(* CODESYS project CANEcho.project

Project tree, tasks and I/O mapping:
  Device : CODESYS Control Win V3, 3S - Smart Software Solutions GmbH, order no. 305021, version 3.5.9.0
    application Application
      libraries: Standard, * (System); CANbus, 3.5.7.0 (3S - Smart Software Solutions GmbH); Common Behaviour Model Library, 0.35.9.0 (3S - Smart Software Solutions GmbH); Time and Date, 3.5.7.0 (3S - Smart Software Solutions GmbH)
      task MainTask (cyclic, interval t#20ms, priority 1) calls PLC_PRG
      program PLC_PRG [ST]
      visualisation Visualization
  text list GlobalTextList
  function block CANEcho [ST]: CyclicAction, CleanupAction, StartAction, ResetAction
*)

// Device/Application/PLC_PRG
PROGRAM PLC_PRG
VAR
	aEchoTest : ARRAY[0..ciEchoInstances-1] OF CANEcho;
	axResetBusAlarm : ARRAY[0..ciEchoInstances-1] OF BOOL;
	i : INT;
	xInit : BOOL;
END_VAR
VAR CONSTANT
	ciEchoInstances : INT := 2;
END_VAR

IF NOT xInit THEN
	FOR i := 0 TO ciEchoInstances - 1 DO
		aEchoTest[i].usiNetID := TO_USINT(i);
	END_FOR
	
	xInit := TRUE;
END_IF

FOR i := 0 TO ciEchoInstances - 1 DO
	aEchoTest[i](xResetBusAlarm := axResetBusAlarm[i]);
END_FOR

END_PROGRAM

// CANEcho
FUNCTION_BLOCK CANEcho EXTENDS CBML.LConC
VAR_INPUT
	usiNetID : USINT;
	wBaudrate : WORD := 1000;
	xSupport29bit : BOOL := TRUE;
	ctTxMessages : CAA.COUNT := 100;
	xMessageDurationTest : BOOL := TRUE;
	dwMessageDurationCOBID : DWORD := 16#701;
END_VAR
VAR_IN_OUT
	xResetBusAlarm : BOOL;
END_VAR
VAR_OUTPUT
	diagInfo : CL2.DIAGNOSIS_INFO;
	udiMessageDurationMinTimeSpan : UDINT := 16#FFFFFFFF;
	udiMessageDurationCurTimeSpan : UDINT;
	udiMessageDurationMaxTimeSpan : UDINT;
END_VAR
VAR
	hDriver : CAA.HANDLE := CAA.gc_hINVALID;
	hReceiver : CAA.HANDLE := CAA.gc_hINVALID;
	eError : CL2.ERROR;
	hRxMsg : CAA.HANDLE := CAA.gc_hINVALID;
	pRxData : POINTER TO CL2I.DATA;
	hTxMsg : CAA.HANDLE := CAA.gc_hINVALID;
	pTxData : POINTER TO CL2I.DATA;
	ctMsgLeft : CAA.COUNT;
	diMsgRecv: DINT;
	i : INT;
	
	cobId : CL2I.COBID;
	usiLen : USINT;
	x29Bit : BOOL;
	xRTR : BOOL;
	xTxFrame : BOOL;
	tkStart : CAA.TICK;
	xLastMessageDurationTest : BOOL;
	
	//Test Mode
	xEchoMessages : BOOL := TRUE;
END_VAR

SUPER^();

METHOD CyclicAction
VAR_INPUT
	itfTimingController	: CBML.ITimingController;
END_VAR
VAR_OUTPUT
	xComplete	: BOOL;
	iErrorID	: INT;
END_VAR
CL2.GetDiagnosis(hDriver, ADR(diagInfo));

{warning disable C0371}
IF xResetBusAlarm THEN
	CL2.ResetBusAlarm(hDriver);
	xResetBusAlarm := FALSE;
END_IF
{warning restore C0371}

IF (xLastMessageDurationTest <> xMessageDurationTest) THEN
	//Reset Heartbeat Test
	tkStart := 0;
	udiMessageDurationMinTimeSpan := 16#FFFFFFFF;
	udiMessageDurationCurTimeSpan := 0;
	udiMessageDurationMaxTimeSpan := 0;
END_IF

xLastMessageDurationTest := xMessageDurationTest;

REPEAT
	hRxMsg := CL2.Read(hReceiverId:=hReceiver, pctMsgLeft:=ADR(ctMsgLeft), peError:=ADR(eError));
	IF hRxMsg <> CAA.gc_hINVALID THEN
		x29Bit := CL2.Is29BitIdMessage(hMessage := hRxMsg, peError := CAA.gc_pNULL);
		xTxFrame := CL2.IsTransmitMessage(hMessage := hRxMsg, peError := CAA.gc_pNULL);
		xRTR := CL2.IsRTRMessage(hMessage := hRxMsg, peError := CAA.gc_pNULL);
		cobId := CL2.GetMessageId(hMessage := hRxMsg, peError:= CAA.gc_pNULL);
		usiLen := CL2.GetMessageLength(hMessage := hRxMsg, peError := CAA.gc_pNULL);
		pRxData := CL2.GetMessageDataPointer(hMessage := hRxMsg, peError := ADR(eError));
		diMsgRecv := diMsgRecv + 1;
		IF xEchoMessages THEN
			IF pRxData <> CAA.gc_pNULL THEN
				//echo message
				hTxMsg := CL2.CreateMessage(
						hDriver:= hDriver, 
						cobID := cobId+1, 
						usiLength := usiLen, 
						xRTR := xRTR, 
						x29BitID := x29Bit, 
						peError := ADR(eError)
				);
					
				IF hTxMsg <> CAA.gc_hINVALID THEN
					pTxData := CL2.GetMessageDataPointer(hMessage := hTxMsg, peError := ADR(eError));
					IF pTxData <> CAA.gc_pNULL AND usiLen <> 0 THEN
						FOR i := 0 TO usiLen - 1 DO
							pTxData^[i] := pRxData^[i];
						END_FOR
					END_IF
					eError := CL2.Write(hDriver:= hDriver, hMessage := hTxMsg, usiPriority := 1, xEnableSyncWindow := FALSE);
					IF eError <> CL2.ERROR.NO_ERROR THEN
						CL2.FreeMessage(hMessage := hTxMsg);
					END_IF
	
					hTxMsg := CAA.gc_hINVALID;
					pTxData := CAA.gc_pNULL;
				END_IF
			END_IF
		END_IF
		
		IF xMessageDurationTest THEN
			IF (cobId = dwMessageDurationCOBID) THEN
				IF (tkStart <> 0) THEN
					udiMessageDurationCurTimeSpan := TICKU.GetElapsedTimeInUSec(tkStart);
					IF (udiMessageDurationCurTimeSpan > udiMessageDurationMaxTimeSpan) THEN
						udiMessageDurationMaxTimeSpan := udiMessageDurationCurTimeSpan;
					ELSIF udiMessageDurationCurTimeSpan < udiMessageDurationMinTimeSpan THEN
						udiMessageDurationMinTimeSpan := udiMessageDurationCurTimeSpan;
					END_IF
				END_IF
				tkStart := TICKS.GetTick(TRUE);
			END_IF
		END_IF
		
		CL2.FreeMessage(hMessage := hRxMsg);
		hRxMsg := CAA.gc_hINVALID;
		pRxData := CAA.gc_pNULL;
	END_IF
UNTIL ctMsgLeft = 0 
END_REPEAT

CL2.GetDiagnosis(hDriver, ADR(diagInfo));
END_METHOD

METHOD CleanupAction
VAR_INPUT
	xAbortProposed	: BOOL;
	iErrorIDProposed	: INT;
END_VAR
VAR_OUTPUT
	xComplete	: BOOL;
	xAbort	: BOOL;
	iErrorID	: INT;
END_VAR
CL2.DeleteReceiver(hReceiverId := hReceiver);
hReceiver := CAA.gc_hINVALID;

CL2.DriverClose(hDriver := hDriver);
hDriver := CAA.gc_hINVALID;

xAbort := xAbortProposed;
iErrorID := iErrorIDProposed;

xComplete := TRUE;
END_METHOD

METHOD StartAction
VAR_OUTPUT
	xComplete	: BOOL;
	iErrorID	: INT;
END_VAR
hDriver:= CL2.DriverOpenH(
	usiNetId :=usiNetID, 
	uiBaudrate := wBaudrate, 
	xSupport29Bits := xSupport29bit, 
	ctMessages := ctTxMessages, 
	peError := ADR(eError)
);

IF hDriver <> CAA.gc_hINVALID THEN
	hReceiver := CL2.CreateMaskReceiver(
		hDriver:= hDriver, 
		cobIdValue := 0, 
		cobIdMask := 0, 
		xRTRValue := 0, 
		xRTRMask := 0, 
		x29BitIdValue := FALSE, 
		x29BitIdMask := NOT xSupport29bit, 
		xTransmitValue := FALSE, 
		xTransmitMask := TRUE, 
		xAlwaysNewest := FALSE, 
		eEvent := CB.EVENT.NO_EVENT, 
		xEnableSyncWindow := FALSE, 
		peError := ADR(eError)
	);
END_IF

IF hDriver = CAA.gc_hINVALID THEN
	iErrorID := 1;
ELSE
	xComplete := TRUE;
END_IF
END_METHOD

METHOD ResetAction
VAR_OUTPUT
	xComplete	: BOOL;
END_VAR
udiMessageDurationMinTimeSpan := 16#FFFFFFFF;
udiMessageDurationCurTimeSpan := 0;
udiMessageDurationMaxTimeSpan := 0;
xLastMessageDurationTest := FALSE;
xComplete := TRUE;
END_METHOD

END_FUNCTION_BLOCK

// Device/Application/Visualization
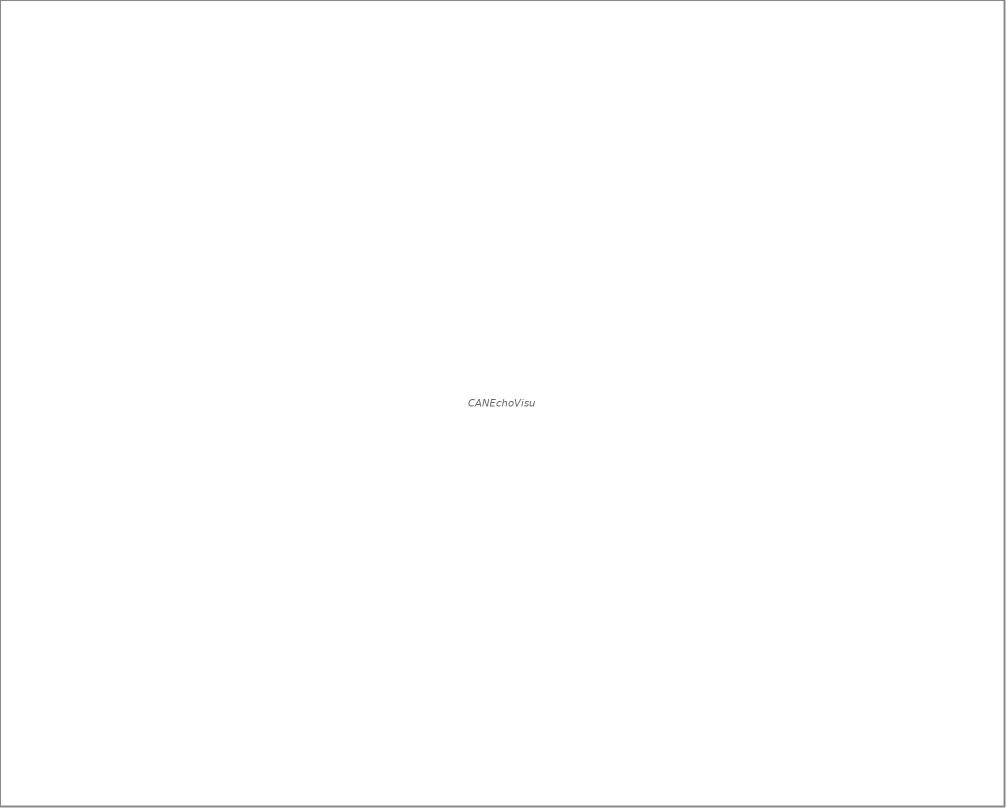
VISUALIZATION Visualization  // 1006x808
    TabControl (0,0 1004x806)
        shows CANEchoVisu(echoFB := PLC_PRG.aEchoTest[0])
        shows CANEchoVisu(echoFB := PLC_PRG.aEchoTest[1])
        [0]: TabTitle=Driver1
        [1]: TabTitle=Driver2
END_VISUALIZATION
